TYPE ST_PrintingBed :
STRUCT
	fSetTemp		: REAL;			// Solltemperatur Druckbett
	fActualTemp		: REAL;			// Isttemperatur Druckbett
	bAtTemp			: BOOL;			// Solltemperatur erreicht (0.5°C Toleranz)
	bErrorReset		: BOOL;
	bError        	: BOOL;			// Fehler
    nErrorID      	: UDINT;
    sErrorMsg 		: STRING(80);
END_STRUCT
END_TYPE

(* stored: Version 1.1.0.1
   DUT ST_PrintingBed: Id {40b7606b-d497-48ff-b6b5-f0d9dac24e3d} *)
